PROGRAM taskDataGrab
VAR
END_VAR

//call the data grab
prgDataGrab();

END_PROGRAM

(* stored: Version 1.1.0.1, ProductVersion 3.1.4024.11
   POU taskDataGrab: Id {7a4f74d7-5fdf-0170-3ab7-66ec9ac5539a}, SpecialFunc None *)
